Yaskawa INFORM job: SET_IDS_FULL.JBI

/JOB
//NAME SET_IDS_FULL
///FOLDERNAME TWINCAT_KOMMUNIKATION
//POS
///NPOS 0,0,0,0,0,0
//ALIAS
///LVARS 0,5,0,0,0,0,0,0
LI000 WID
LI001 NAHT
LI002 LAGE
LI003 RAUPE
LI004 SCHW
//ARGINFO
///ARGTYPE I,I,I,I,I,,,
///COMMENT
WID
NAHT
LAGE
RAUPE
SCHW



//INST
///DATE 2023/05/03 17:27
///COMM SET WID AND NUMBERS
///ATTR SC,RW
///LVARS 0,5,0,0,0,0,0,0
NOP
'--------------------------------
'Dieser Job setzt einen
'vollständigen Satz an ID-Nummern
'mit WID
'--------------------------------
'Argumente lesen
GETARG WID IARG#(1)
GETARG NAHT IARG#(2)
GETARG LAGE IARG#(3)
GETARG RAUPE IARG#(4)
GETARG SCHW IARG#(5)
'--------------------------------
'ID Trigger festsetzen
SETREG MREG#(69) 1
'--------------------------------
'WID setzen
CALL JOB:SET_ID ARGFWID ARGF"WID"
'--------------------------------
'Nummern setzen
CALL JOB:SET_IDS ARGFNAHT ARGFLAGE ARGFRAUPE ARGFSCHW
'--------------------------------
'ID Trigger freigeben
SETREG MREG#(69) 0
END
